VAR_GLOBAL
	AufzugSensorEinlaufFoerderband	:	BOOL;
	AufzugSensorAuslaufFoerderband	:	BOOL;
	AufzugFoerderbandVorwaerts	:	BOOL;
	AufzugFoerderbandRueckwaerts	:	BOOL;
	AufzugSollwert	:	WORD;
	AufzugIstwert	:	WORD;
	
	(*======================= Simulation* =======================*)
	IstPositionConverted	:	REAL;
	SollPosition	:	REAL;
	AufzugInPosition	:	BOOL;
	AufzugBewegen	:	BOOL;
	AufzugFoerderbandVor	: BOOL;
	AufzugFoerderbandRueck	: BOOL;
	AufzugFoerderbandStop	: BOOL;
	instFBElevator	:	FB_Elevator;
END_VAR

(* stored: Version 1.1.0.1
   GVL Elevator: Id {4fe7e48e-4868-4340-aa32-2af6f80c9da8} *)
